FUNCTION_BLOCK Timer_TON_2 (* Composite Function Block Type *)
  (* Standard: 61499-2 *)
  (* Version 0.0, 5/24/2016, gulzha, nxtControl GmbH, template *)
  PACKAGE Main;
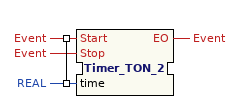
  EVENT_INPUT
    Start WITH time;
    Stop;
  END_EVENT
  EVENT_OUTPUT
    EO; (* Periodic event at period DT,starting at DT after START *)
  END_EVENT
  VAR_INPUT
    time : REAL; (* in seconds *)
  END_VAR
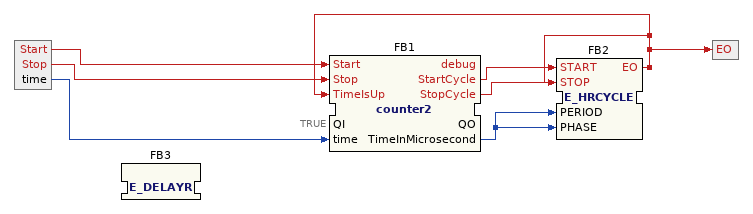
  FBS
    FB2 : E_HRCYCLE;
    FB1 : counter2(QI := TRUE);
    FB3 : E_DELAYR;
  END_FBS
  EVENT_CONNECTIONS
    FB1.StartCycle TO FB2.START;
    FB1.StopCycle TO FB2.STOP;
    Start TO FB1.Start;
    Stop TO FB1.Stop;
    FB2.EO TO FB1.TimeIsUp;
    FB2.EO TO EO;
    FB2.EO TO FB2.STOP;
  END_CONNECTIONS
  DATA_CONNECTIONS
    FB1.TimeInMicrosecond TO FB2.PERIOD;
    time TO FB1.time;
    FB1.TimeInMicrosecond TO FB2.PHASE;
  END_CONNECTIONS
END_FUNCTION_BLOCK
